FUNCTION_BLOCK FB_TrafficLightConsumer
VAR
    light : B3TrafficLight_Plc.FB_TrafficLight;
    lastState : INT;
END_VAR

lastState := light.Step();

END_FUNCTION_BLOCK

(* stored: Version 1.1.0.1
   POU FB_TrafficLightConsumer: Id {395df02d-4da9-44f7-9319-21dab7856a58}, SpecialFunc None *)
